PROGRAM MAIN
VAR
END_VAR

END_PROGRAM

(* stored: Version 1.1.0.1
   POU MAIN: Id {68e6d7cc-dbce-4f85-9bb2-85846695a555} *)
